FUNCTION_BLOCK Horse_Object EXTENDS TcoCore.TcoObject
VAR
	_price	: LREAL;	
END_VAR

PROPERTY Price : LREAL
GET
Price := _price;
END_GET
SET
_price := Price;
END_SET
END_PROPERTY

END_FUNCTION_BLOCK

(* stored: Version 1.1.0.1, ProductVersion 3.1.4024.6
   POU Horse_Object: Id {318d333c-8793-0528-10f0-90d7a7341f0d}, SpecialFunc None
   Property Price: Id {e3ea7672-3134-0a22-002f-336efed6f2c1}
   Get Get: Id {60034efa-7b3c-067d-33aa-263f0b37071f}
   Set Set: Id {2a4ab36a-6675-009d-23bc-d597f5ec2ca8} *)
